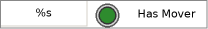
VISUALIZATION V_Station  // 208x29
VAR_IN_OUT
	Station : ST_Station_HMI;
END_VAR
    Textfield (0,0 87x26), "%s", text variable: Station.Status.MoverID
    Lamp1 (92,2 31x27), variable: Station.Status.HasMover, style: Lamp-Lamp1-Green
    Textfield (125,1 83x26), "Has Mover"
END_VISUALIZATION

(* stored: Version 1.1.0.1, ProductVersion 3.1.4024.12
   Visu V_Station: Id {4c4b21d7-a44e-4700-a247-979fce7e4dc2} *)
